// TIA Portal project "LMU02_HMI" (V16)
// HMI for lolly machine upgrade. Communcation is over Modbus TCP/IP.

(* hardware
DEVICE "HMI_1"  KTP600 Basic color PN Portrait
   slot 0: "HMI_1"  KTP600 Basic color PN Portrait  6AV6 647-0AD11-3AX0  12.0.0.0
   slot 1: "HMI_RT_1"  KTP600 Basic color PN Portrait  6AV6 647-0AD11-3AX0  12.0.0.0
   slot 5: "HMI_1.IE_CP_1"  PROFINET Interface  12.0.0.0
      slot 1: "PROFINET Interface_1"  PROFINET Interface
         slot 1: "Port_1"  Port
*)

(* ===== HMI "HMI_RT_1" =====
system functions are stored by id; their names below are inferred from use
connection "Modbus": ETHERNET, SMART_MODBUS_TCP

HMI tags "Default tag table"
   "Tag_ScreenNumber" : UInt, internal
   "start" : Bit AT 0x16688, 1 s
   "stop" : Bit AT 0x16689, 1 s
   "manual" : Bit AT 0x16690, 1 s
   "sortAll" : Bit AT 0x16691, 1 s
   "dumpAll" : Bit AT 0x16692, 1 s
   "leaveEmpty" : Bit AT 0x16693, 1 s
   "hopperRefilled" : Bit AT 0x16694, 1 s
   "okThanks" : Bit AT 0x16695, 1 s
   "errorAck" : Bit AT 0x16695, 1 s
   "V0_write" : Bit AT 0x16705, 1 s
   "V1_write" : Bit AT 0x16706, 1 s
   "V2_write" : Bit AT 0x16707, 1 s
   "V3_write" : Bit AT 0x16708, 1 s
   "V4_write" : Bit AT 0x16709, 1 s
   "V5_write" : Bit AT 0x16710, 1 s
   "V6_write" : Bit AT 0x16711, 1 s
   "V7_write" : Bit AT 0x16712, 1 s
   "V8_write" : Bit AT 0x16713, 1 s
   "V9_write" : Bit AT 0x16714, 1 s
   "V10_write" : Bit AT 0x16715, 1 s
   "V11_write" : Bit AT 0x16716, 1 s
   "V0_read" : Bit AT 0x16609, 1 s
   "V1_read" : Bit AT 0x16610, 1 s
   "V2_read" : Bit AT 0x16611, 1 s
   "V3_read" : Bit AT 0x16612, 1 s
   "V4_read" : Bit AT 0x16613, 1 s
   "V5_read" : Bit AT 0x16614, 1 s
   "V6_read" : Bit AT 0x16615, 1 s
   "V7_read" : Bit AT 0x16624, 1 s
   "V8_read" : Bit AT 0x16625, 1 s
   "V9_read" : Bit AT 0x16626, 1 s
   "V10_read" : Bit AT 0x16627, 1 s
   "V11_read" : Bit AT 0x16628, 1 s
   "S01" : Bit AT 0x16589, 1 s
   "S02" : Bit AT 0x16590, 1 s
   "S11" : Bit AT 0x16595, 1 s
   "S12" : Bit AT 0x16596, 1 s
   "S21" : Bit AT 0x16597, 1 s
   "S22" : Bit AT 0x16598, 1 s
   "S31" : Bit AT 0x16599, 1 s
   "S32" : Bit AT 0x16600, 1 s
   "S41" : Bit AT 0x16585, 1 s
   "S42" : Bit AT 0x16586, 1 s
   "S51" : Bit AT 0x16587, 1 s
   "S52" : Bit AT 0x16588, 1 s
   "S61" : Bit AT 0x16591, 1 s
   "S62" : Bit AT 0x16592, 1 s
   "S71" : Bit AT 0x16593, 1 s
   "S72" : Bit AT 0x16594, 1 s
   "S81" : Bit AT 0x16601, 1 s
   "S82" : Bit AT 0x16602, 1 s
   "S91" : Bit AT 0x16603, 1 s
   "S92" : Bit AT 0x16604, 1 s
   "P1" : Bit AT 0x16605, 1 s
   "P2" : Bit AT 0x16606, 1 s
   "C1" : Bit AT 0x16616, 1 s
   "C2" : Bit AT 0x16617, 1 s
   "C3" : Bit AT 0x16618, 1 s
   "C4" : Bit AT 0x16619, 1 s

Template "Template_1" 240x320
   Button "Start screen" at 202,57 size 37x52; TextOff 'Start screen'; PictureOff "NavigateHome_KTP600_Basic_color_PN_Portrait"; PictureOn "NavigateHome_KTP600_Basic_color_PN_Portrait"
      on Release: ActivateScreen("1_Home", 0)
   Button "Template_Button" at 202,109 size 37x52; TextOff 'IO'; TextOn 'MEOW'; PictureOff "manual"
      on Release: ActivateScreen("2_Manual", 0)
   Button "Template_Button_1" at 202,161 size 37x52; TextOff 'IO'
      on Release: ActivateScreen("3_IOA", 0)
   Button "Alarms" at 202,213 size 37x52; TextOff 'Alarms'; PictureOff "AlarmDisplay_KTP600_Basic_color_PN_Portrait"; PictureOn "AlarmDisplay_KTP600_Basic_color_PN_Portrait"
      on Release: function_ef3f5d25("Alarm window_Unacknowledged", -1)
   Button "Exit" at 202,266 size 37x52; TextOff 'Exit'; PictureOff "ExitRuntime_KTP600_Basic_color_PN_Portrait"; PictureOn "ExitRuntime_KTP600_Basic_color_PN_Portrait"
      on Release: StopRuntime(0)
   SymbolicIOField "Symbolic_IO_Field_Screen" at 48,5 size 98x20; TextOff '0'; TextOn '1'; TextList "TextList_ScreenNames"
      ProcessValue <- "Tag_ScreenNumber"
      on Change: ActivateScreenByNumber("Tag_ScreenNumber", 0)
   DateTimeField "HmiScreenItemData" at 155,15 size 85x15
   DateTimeField "HmiScreenItemData_1" at 155,0 size 85x15
   GraphicView "Template_Graphic view_1" at 34,288 size 138x30; Picture "Graphic_3"
   Softkey "Softkey_F6" at 0,0 size 0x0
      on KeyUp: ActivateScreen("1_Home", 0)

screen "1_Home" 240x320, template "Template_1"
   on GenerateScreen: SetTag("Tag_ScreenNumber", 1)
   Button "Template_Button_2" at 12,43 size 54x32; TextOff 'Start'
   Button "Template_Button_3" at 13,91 size 53x32; TextOff 'Sort All'
   Group "Group" at 115,169 size 45x36
   Group "Group_1" at 115,126 size 45x36
   Group "Group_2" at 115,83 size 45x36
   Group "Group_3" at 115,40 size 45x36
   Button "Template_Button_4" at 13,140 size 53x32; TextOff 'Dump All'
   Button "Template_Button_1" at 13,188 size 53x32; TextOff 'Manual'
   Button "Template_Button_5" at 13,237 size 53x32; TextOff 'Stop'
   IOField "Template_I/O field_4" at 116,182 size 22x23; FormatPattern 9
   TextField "Template_Text field_4" at 115,169 size 45x13; Text 'Colour 4'
   IOField "Template_I/O field_3" at 116,139 size 22x23; FormatPattern 9
   TextField "Template_Text field_3" at 115,126 size 45x13; Text 'Colour 3'
   IOField "Template_I/O field_2" at 116,96 size 22x23; FormatPattern 9
   TextField "Template_Text field_2" at 115,83 size 45x13; Text 'Colour 2'
   IOField "Template_I/O field_1" at 116,53 size 22x23; FormatPattern 9
   TextField "Template_Text field_1" at 115,40 size 45x13; Text 'Colour 1'

screen "2_Manual" 240x320, template "Template_1"
   on GenerateScreen: SetTag("Tag_ScreenNumber", 2)
   Button "Button_1" at 14,40 size 32x32; TextOff 'V0'
      on Click: InvertBit("V0_write")
   Button "Button_2" at 14,81 size 32x32; TextOff 'V1'
      on Click: InvertBit("V1_write")
   Button "Button_3" at 14,123 size 32x32; TextOff 'V2'
      on Click: InvertBit("V2_write")
   Button "Button_4" at 14,164 size 32x32; TextOff 'V3'
      on Click: InvertBit("V3_write")
   Button "Button_5" at 14,206 size 32x32; TextOff 'V4'
      on Click: InvertBit("V4_write")
   Button "Button_6" at 14,248 size 32x32; TextOff 'V5'
      on Click: InvertBit("V5_write")
   Button "Button_7" at 102,40 size 32x32; TextOff 'V6'
      on Click: InvertBit("V6_write")
   Button "Button_8" at 102,81 size 32x32; TextOff 'V7'
      on Click: InvertBit("V7_write")
   Button "Button_9" at 102,123 size 32x32; TextOff 'V8'
      on Click: InvertBit("V8_write")
   Button "Button_10" at 102,164 size 32x32; TextOff 'V9'
      on Click: InvertBit("V9_write")
   Button "Button_11" at 102,206 size 32x32; TextOff 'V10'
      on Click: InvertBit("V10_write")
   Button "Button_12" at 102,248 size 32x32; TextOff 'V11'
      on Click: InvertBit("V11_write")
   TextField "Text field_1" at 49,48 size 34x13; Text 'Reject'
   TextField "Text field_2" at 49,90 size 46x13; Text 'Top Pad.'
   TextField "Text field_3" at 50,132 size 53x13; Text 'Right Pad.'
   TextField "Text field_4" at 49,174 size 47x13; Text 'Left Pad.'
   TextField "Text field_5" at 49,216 size 36x13; Text 'Drop 1'
   TextField "Text field_6" at 50,258 size 36x13; Text 'Drop 2'
   TextField "Text field_7" at 141,48 size 45x13; Text 'Colour 4'
   TextField "Text field_8" at 141,90 size 45x13; Text 'Colour 3'
   TextField "Text field_9" at 141,132 size 45x13; Text 'Colour 2'
   TextField "Text field_10" at 141,174 size 45x13; Text 'Colour 1'
   TextField "Text field_11" at 141,216 size 46x13; Text 'Dispense'
   TextField "Text field_12" at 141,258 size 36x13; Text 'Return'

screen "Project information" 240x320, template "Template_1"
   on GenerateScreen: SetTag("Tag_ScreenNumber", 10)
   TextField "HmiScreenItemData" at 4,63 size 194x20; Text 'Project name:'
   TextField "HmiScreenItemData_1" at 4,84 size 194x20; Text 'lollyMachineUpgrade_HMI'
   TextField "HmiScreenItemData_2" at 4,105 size 194x20; Text 'Created on:'
   TextField "HmiScreenItemData_3" at 4,126 size 194x20; Text '8/19/2022 9:08:58 AM'
   TextField "HmiScreenItemData_4" at 4,147 size 194x20; Text 'Author:'
   TextField "HmiScreenItemData_5" at 4,168 size 194x20; Text 'Henry Davies'
   TextField "HmiScreenItemData_6" at 4,189 size 194x20; Text 'Description:'
   TextField "HmiScreenItemData_7" at 4,210 size 194x20; Text 'HMI for lolly machine upgrade. Communcation is over Modbus TCP/IP.'

screen "System information" 240x320, template "Template_1"
   on GenerateScreen: SetTag("Tag_ScreenNumber", 11)
   TextField "HmiScreenItemData" at 4,63 size 194x20; Text 'HMI device type:'
   TextField "HmiScreenItemData_1" at 4,84 size 194x20; Text 'KTP600 Basic color PN Portrait 12.0'
   TextField "HmiScreenItemData_2" at 4,105 size 194x20; Text 'Connection:'
   TextField "HmiScreenItemData_3" at 4,126 size 194x20; Text '(not configured)'
   TextField "HmiScreenItemData_4" at 4,147 size 194x20; Text 'PLC:'
   TextField "HmiScreenItemData_5" at 4,168 size 194x20; Text '<PLC>'

screen "3_IOA" 240x320, template "Template_1"
   on GenerateScreen: SetTag("Tag_ScreenNumber", 3)
   TextField "Text field_1" at 11,40 size 16x13; Text 'V0'
   TextField "Text field_2" at 11,60 size 16x13; Text 'V1'
   TextField "Text field_3" at 11,80 size 16x13; Text 'V2'
   TextField "Text field_4" at 11,101 size 16x13; Text 'V3'
   TextField "Text field_5" at 11,121 size 16x13; Text 'V4'
   TextField "Text field_6" at 11,141 size 16x13; Text 'V5'
   TextField "Text field_7" at 11,162 size 16x13; Text 'V6'
   TextField "Text field_8" at 11,182 size 16x13; Text 'V7'
   TextField "Text field_9" at 11,202 size 16x13; Text 'V8'
   TextField "Text field_10" at 11,223 size 16x13; Text 'V9'
   TextField "Text field_11" at 11,243 size 23x13; Text 'V10'
   TextField "Text field_12" at 11,264 size 23x13; Text 'V11'
   Circle "Circle_1" at 35,41 size 12x12
      Appearance <- "V0_read"
   TextField "Text field_13" at 65,40 size 22x13; Text 'S01'
   TextField "Text field_14" at 118,40 size 22x13; Text 'S02'
   Button "Button_1" at 64,246 size 90x27; TextOff 'Next'
      on Release: ActivateScreen("4_IOB", 0)
   TextField "Text field_15" at 65,60 size 22x13; Text 'S11'
   TextField "Text field_16" at 118,60 size 22x13; Text 'S12'
   TextField "Text field_17" at 65,80 size 22x13; Text 'S21'
   TextField "Text field_18" at 118,80 size 22x13; Text 'S22'
   TextField "Text field_19" at 65,101 size 22x13; Text 'S31'
   TextField "Text field_20" at 118,101 size 22x13; Text 'S32'
   TextField "Text field_21" at 65,121 size 22x13; Text 'S41'
   TextField "Text field_22" at 118,121 size 22x13; Text 'S42'
   TextField "Text field_23" at 65,141 size 22x13; Text 'S51'
   TextField "Text field_24" at 118,141 size 22x13; Text 'S52'
   TextField "Text field_25" at 65,162 size 22x13; Text 'S61'
   TextField "Text field_26" at 118,162 size 22x13; Text 'S62'
   TextField "Text field_27" at 65,182 size 22x13; Text 'S71'
   TextField "Text field_28" at 118,182 size 22x13; Text 'S72'
   TextField "Text field_29" at 65,202 size 22x13; Text 'S81'
   TextField "Text field_30" at 118,202 size 22x13; Text 'S82'
   TextField "Text field_31" at 65,223 size 22x13; Text 'S91'
   TextField "Text field_32" at 118,223 size 22x13; Text 'S92'
   Circle "Circle_2" at 35,61 size 12x12
      Appearance <- "V1_read"
   Circle "Circle_3" at 35,81 size 12x12
      Appearance <- "V2_read"
   Circle "Circle_4" at 35,102 size 12x12
      Appearance <- "V3_read"
   Circle "Circle_5" at 35,122 size 12x12
      Appearance <- "V4_read"
   Circle "Circle_6" at 35,142 size 12x12
      Appearance <- "V5_read"
   Circle "Circle_7" at 35,163 size 12x12
      Appearance <- "V6_read"
   Circle "Circle_8" at 35,183 size 12x12
      Appearance <- "V7_read"
   Circle "Circle_9" at 35,203 size 12x12
      Appearance <- "V8_read"
   Circle "Circle_10" at 35,224 size 12x12
      Appearance <- "V9_read"
   Circle "Circle_11" at 35,244 size 12x12
      Appearance <- "V10_read"
   Circle "Circle_12" at 35,265 size 12x12
      Appearance <- "V11_read"
   Circle "Circle_13" at 87,41 size 12x12
      Appearance <- "S01"
   Circle "Circle_14" at 87,61 size 12x12
      Appearance <- "S11"
   Circle "Circle_15" at 87,81 size 12x12
      Appearance <- "S21"
   Circle "Circle_16" at 87,102 size 12x12
      Appearance <- "S31"
   Circle "Circle_17" at 87,122 size 12x12
      Appearance <- "S41"
   Circle "Circle_18" at 87,142 size 12x12
      Appearance <- "S51"
   Circle "Circle_19" at 87,163 size 12x12
      Appearance <- "S61"
   Circle "Circle_20" at 87,183 size 12x12
      Appearance <- "S71"
   Circle "Circle_21" at 87,203 size 12x12
      Appearance <- "S81"
   Circle "Circle_22" at 87,224 size 12x12
      Appearance <- "S91"
   Circle "Circle_23" at 143,41 size 12x12
      Appearance <- "S02"
   Circle "Circle_24" at 143,61 size 12x12
      Appearance <- "S12"
   Circle "Circle_25" at 143,81 size 12x12
      Appearance <- "S22"
   Circle "Circle_26" at 143,102 size 12x12
      Appearance <- "S32"
   Circle "Circle_27" at 143,122 size 12x12
      Appearance <- "S42"
   Circle "Circle_28" at 143,142 size 12x12
      Appearance <- "S52"
   Circle "Circle_29" at 143,163 size 12x12
      Appearance <- "S62"
   Circle "Circle_30" at 143,183 size 12x12
      Appearance <- "S72"
   Circle "Circle_31" at 143,203 size 12x12
      Appearance <- "S82"
   Circle "Circle_32" at 143,224 size 12x12
      Appearance <- "S92"

screen "4_IOB" 240x320, template "Template_1"
   on GenerateScreen: SetTag("Tag_ScreenNumber", 4)
   TextField "Text field_1" at 11,40 size 16x13; Text 'C1'
   TextField "Text field_2" at 11,60 size 16x13; Text 'C2'
   TextField "Text field_3" at 11,80 size 16x13; Text 'C3'
   TextField "Text field_4" at 11,101 size 16x13; Text 'C4'
   TextField "Text field_5" at 11,121 size 16x13; Text 'P1'
   TextField "Text field_6" at 11,141 size 16x13; Text 'P2'
   Circle "Circle_1" at 35,41 size 12x12
      Appearance <- "C1"
   Button "Button_1" at 64,246 size 90x27; TextOff 'Previous'
      on Release: ActivateScreen("4_IOB", 0)
   Circle "Circle_2" at 35,61 size 12x12
      Appearance <- "C2"
   Circle "Circle_3" at 35,81 size 12x12
      Appearance <- "C3"
   Circle "Circle_4" at 35,102 size 12x12
      Appearance <- "C4"
   Circle "Circle_5" at 35,122 size 12x12
      Appearance <- "P1"
   Circle "Circle_6" at 35,142 size 12x12
      Appearance <- "P2"
*)